FUNCTION_BLOCK FB_ComponentTest EXTENDS TcUnit.FB_TestSuite
VAR
END_VAR


T01_TestCreateAndLinkData ();

METHOD PRIVATE T01_TestCreateAndLinkData
VAR_INPUT
END_VAR

VAR
	bWynik: BOOL;
END_VAR
IF (TcUnit.TEST_ORDERED ('T01_TestCreateAndLinkData')) THEN
	bWynik := GVL_Variable.fbComponent_1.LinkData (stCommonData := gvl.stCommonData);
	AssertTrue (Condition := bWynik, Message := 'T01 - test linkowania zmiennych ');
	GVL_VariableHMI.fbComponentHMI_1.LinkData (stCommonData := GVL.stCommonData);
	AssertTrue (Condition := bWynik, Message := 'T02 - test linkowania zmiennych ');
	
	
	TcUnit.TEST_FINISHED ();
END_IF
END_METHOD

END_FUNCTION_BLOCK

(* stored: Version 1.1.0.1, ProductVersion 3.1.4024.15
   POU FB_ComponentTest: Id {3cbac2ab-f33e-495d-b5c8-b7ba1b9f5011}, SpecialFunc None
   Method T01_TestCreateAndLinkData: Id {d3c385be-3c77-42c2-89b9-e1b9a0939a42} *)
